Omron CX-Programmer project NewProject (CX-Programmer 9.75)

# PLC NewPLC1: CJ2M CPU11

## Program NewProgram1 (cyclic task 0)
Local symbols
Alarm_Out 100.01 BOOL  ; Drive alarm output
Alarm_Siren 100.03 BOOL  ; Alarm siren
Always_ON A200.00 BOOL  ; Always ON relay
Auto_Mode W0.01 BOOL  ; Auto mode active
Auto_Mode_SW 0.04 BOOL  ; Auto selector switch
Comm_Error W0.03 BOOL  ; Modbus comm fault
EStop_OK 0.03 BOOL  ; Emergency stop healthy
Fault_Active W0.02 BOOL  ; fault active
Fault_Code D301 INT  ; VFD fault code
Fault_Detected W0.04 BOOL  ; fault detected
Fault_Lamp 100.01 BOOL  ; Fault indicator
Fault_Latched W0.03 BOOL
Fault_Reset_PB 0.02 BOOL  ; Fault reset pushbutton
First_Scan A202.00 BOOL  ; First PLC scan
Manual_Mode W0.11 BOOL  ; Manual mode active
Manual_Mode_SW 0.05 BOOL  ; Manual selector switch
Modbus_Busy W0.06 BOOL  ; PMCR active
Motor_OL 0.06 BOOL  ; Motor overload input
Motor_Run_Out 100.00 BOOL  ; Output to VFD run terminal
Run_Command W0.00 BOOL  ; internal run latch
Run_Lamp 100.02 BOOL  ; Run indicator
Speed_Scaled D200 INT  ; 0 -5000 scaling
Speed_Set_Hz D100 INT  ; Speed from HMI
Start_PB 0.00 BOOL  ; Start pushbutton
Status_Word D300 INT  ; VFD status
Stop_PB 0.01 BOOL  ; Stop pushbutton
System_Healthy W0.05 BOOL  ; System healthy
Temp_Hz D150 INT  ; Temporary speed
VFD_Run_FB 0.07 BOOL

### Section Section1

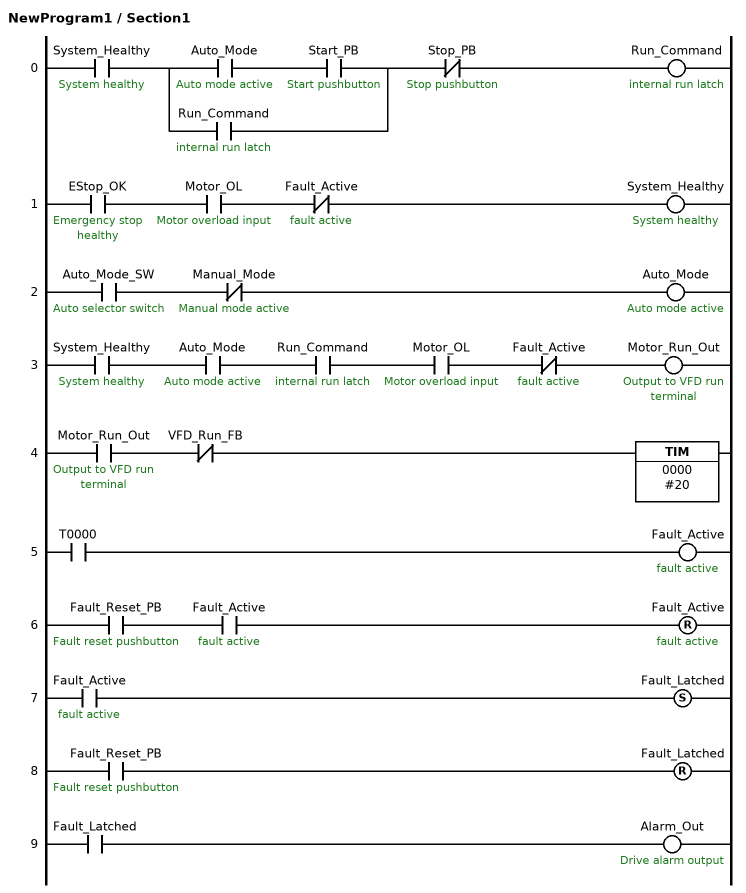
; rung 0
LD System_Healthy  ; System healthy
LD Auto_Mode  ; Auto mode active
AND Start_PB  ; Start pushbutton
OR Run_Command  ; internal run latch
ANDLD
ANDNOT Stop_PB  ; Stop pushbutton
OUT Run_Command  ; internal run latch
; rung 1
LD EStop_OK  ; Emergency stop healthy
AND Motor_OL  ; Motor overload input
ANDNOT Fault_Active  ; fault active
OUT System_Healthy  ; System healthy
; rung 2
LD Auto_Mode_SW  ; Auto selector switch
ANDNOT Manual_Mode  ; Manual mode active
OUT Auto_Mode  ; Auto mode active
; rung 3
LD System_Healthy  ; System healthy
AND Auto_Mode  ; Auto mode active
AND Run_Command  ; internal run latch
AND Motor_OL  ; Motor overload input
ANDNOT Fault_Active  ; fault active
OUT Motor_Run_Out  ; Output to VFD run terminal
; rung 4
LD Motor_Run_Out  ; Output to VFD run terminal
ANDNOT VFD_Run_FB
TIM 0000 #20
; rung 5
LD T0000
OUT Fault_Active  ; fault active
; rung 6
LD Fault_Reset_PB  ; Fault reset pushbutton
AND Fault_Active  ; fault active
RSET Fault_Active  ; fault active
; rung 7
LD Fault_Active  ; fault active
SET Fault_Latched
; rung 8
LD Fault_Reset_PB  ; Fault reset pushbutton
RSET Fault_Latched
; rung 9
LD Fault_Latched
OUT Alarm_Out  ; Drive alarm output

### Section END
; rung 0
END(001)